(* Logix 5000 project; controller APM_Sopladora Emulate 5570 rev 32.11; software revision 32.00 *)

TASK MainTask (continuous, watchdog 500 ms) : MainProgram

MODULES
   Local : Emulate 5570 (ICP 2, rev 32.11)
END_MODULES

VAR_GLOBAL   (* controller tags *)
   A_AbrirMoldes : BOOL;
   A_BandaSopladora : BOOL;
   A_Bandeja : BOOL;
   A_BrazoEx : BOOL;
   A_Grib : BOOL;
   A_Piston : BOOL;
   Aux_Grib : BOOL;
   Aux_Puerta : BOOL;
   BaGF : BOOL;
   BaGF_Ok : BOOL;
   BaGR : BOOL;
   BaGR_Ok : BOOL;
   BaMF : BOOL;
   BaMF_Ok : BOOL;
   BaMR : BOOL;
   BaMR_Ok : BOOL;
   CA_BorrarBotPre : BOOL;
   CA_BotFin : BOOL;
   CA_BotPre : BOOL;
   Count : COUNTER := (PRE := 5);
   Etapa1 : BOOL;
   Etapa10 : BOOL;
   Etapa11 : BOOL;
   Etapa12 : BOOL;
   Etapa13 : BOOL;
   Etapa1A : BOOL;
   Etapa2 : BOOL;
   Etapa2A : BOOL;
   Etapa3 : BOOL;
   Etapa4 : BOOL;
   Etapa5 : BOOL;
   Etapa6 : BOOL;
   Etapa7 : BOOL;
   Etapa8 : BOOL;
   Etapa9 : BOOL;
   Etapa9A : BOOL;
   ND_Start : BOOL;
   ND_Stop : BOOL;
   S_BandejaAtras : BOOL;
   S_BandejaFrente : BOOL;
   S_BotAtGrip : BOOL;
   S_BotAtMolde : BOOL;
   S_BrazoExtendido : BOOL;
   S_BrazoRecogido : BOOL;
   S_PistonAbajo : BOOL;
   S_PistonArriba : BOOL;
   S_PuertaAbierta : BOOL;
   S_PuertaCerrada : BOOL;
   S_Salida : BOOL;
   Sal : BOOL;
   Sal_Ok : BOOL;
   Sec : BOOL;
   Timer1 : TIMER := (PRE := 5000);
   Timer2 : TIMER := (PRE := 3000);
   Timer3 : TIMER := (PRE := 4000);
END_VAR

PROGRAM MainProgram   (* main routine MainRoutine *)

ROUTINE MainRoutine   (* ladder *)
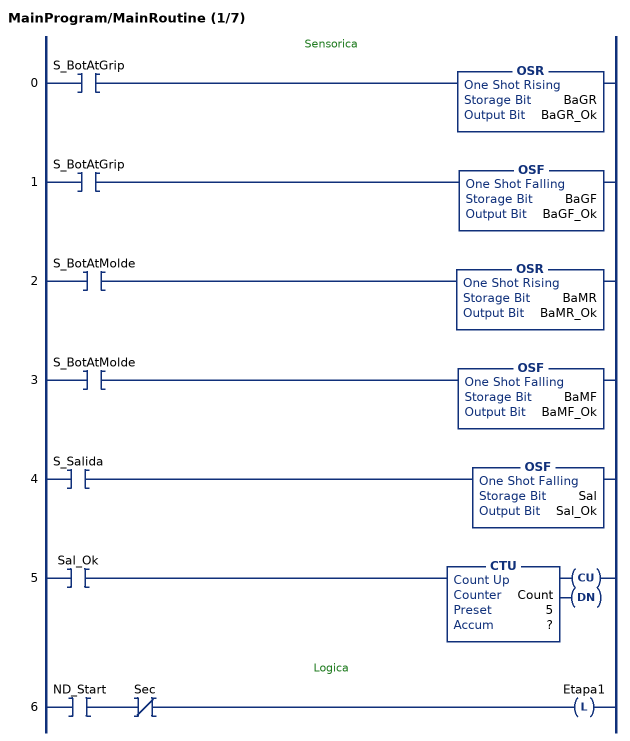
   // Sensorica
   0: XIC(S_BotAtGrip)OSR(BaGR,BaGR_Ok);
   1: XIC(S_BotAtGrip)OSF(BaGF,BaGF_Ok);
   2: XIC(S_BotAtMolde)OSR(BaMR,BaMR_Ok);
   3: XIC(S_BotAtMolde)OSF(BaMF,BaMF_Ok);
   4: XIC(S_Salida)OSF(Sal,Sal_Ok);
   5: XIC(Sal_Ok)CTU(Count,?,?);
   // Logica
   6: XIC(ND_Start)XIO(Sec)OTL(Etapa1);
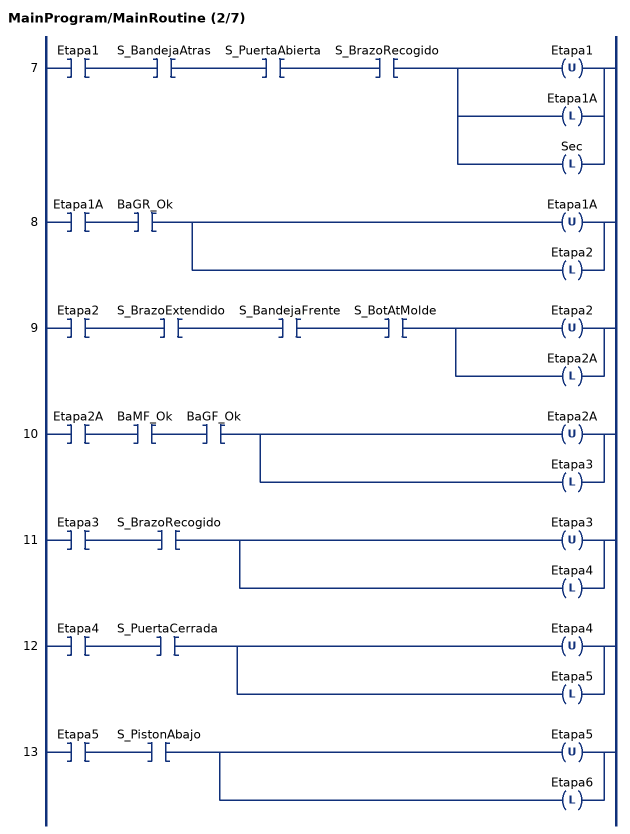
   7: XIC(Etapa1)XIC(S_BandejaAtras)XIC(S_PuertaAbierta)XIC(S_BrazoRecogido)[OTU(Etapa1) ,[OTL(Etapa1A) ,OTL(Sec) ] ];
   8: XIC(Etapa1A)XIC(BaGR_Ok)[OTU(Etapa1A) ,OTL(Etapa2) ];
   9: XIC(Etapa2)XIC(S_BrazoExtendido)XIC(S_BandejaFrente)XIC(S_BotAtMolde)[OTU(Etapa2) ,OTL(Etapa2A) ];
   10: XIC(Etapa2A)XIC(BaMF_Ok)XIC(BaGF_Ok)[OTU(Etapa2A) ,OTL(Etapa3) ];
   11: XIC(Etapa3)XIC(S_BrazoRecogido)[OTU(Etapa3) ,OTL(Etapa4) ];
   12: XIC(Etapa4)XIC(S_PuertaCerrada)[OTU(Etapa4) ,OTL(Etapa5) ];
   13: XIC(Etapa5)XIC(S_PistonAbajo)[OTU(Etapa5) ,OTL(Etapa6) ];
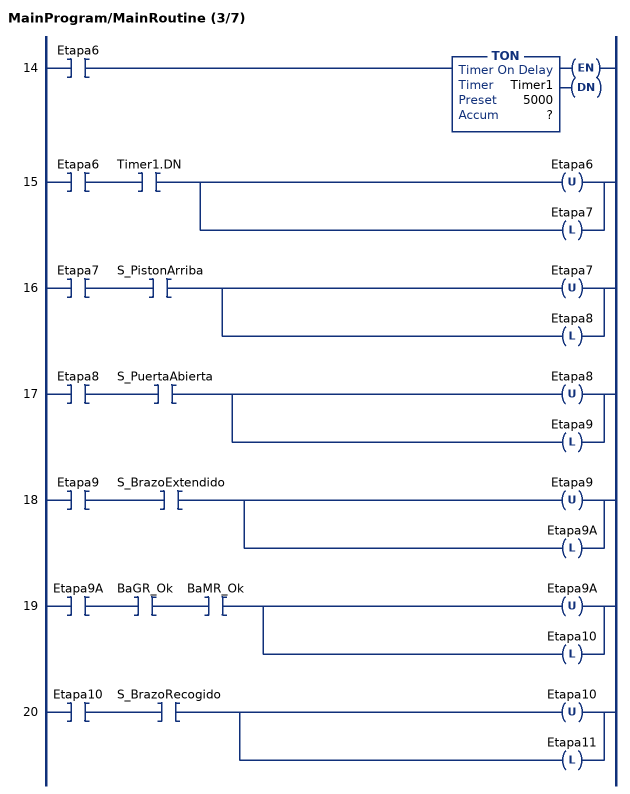
   14: XIC(Etapa6)TON(Timer1,?,?);
   15: XIC(Etapa6)XIC(Timer1.DN)[OTU(Etapa6) ,OTL(Etapa7) ];
   16: XIC(Etapa7)XIC(S_PistonArriba)[OTU(Etapa7) ,OTL(Etapa8) ];
   17: XIC(Etapa8)XIC(S_PuertaAbierta)[OTU(Etapa8) ,OTL(Etapa9) ];
   18: XIC(Etapa9)XIC(S_BrazoExtendido)[OTU(Etapa9) ,OTL(Etapa9A) ];
   19: XIC(Etapa9A)XIC(BaGR_Ok)XIC(BaMR_Ok)[OTU(Etapa9A) ,OTL(Etapa10) ];
   20: XIC(Etapa10)XIC(S_BrazoRecogido)[OTU(Etapa10) ,OTL(Etapa11) ];
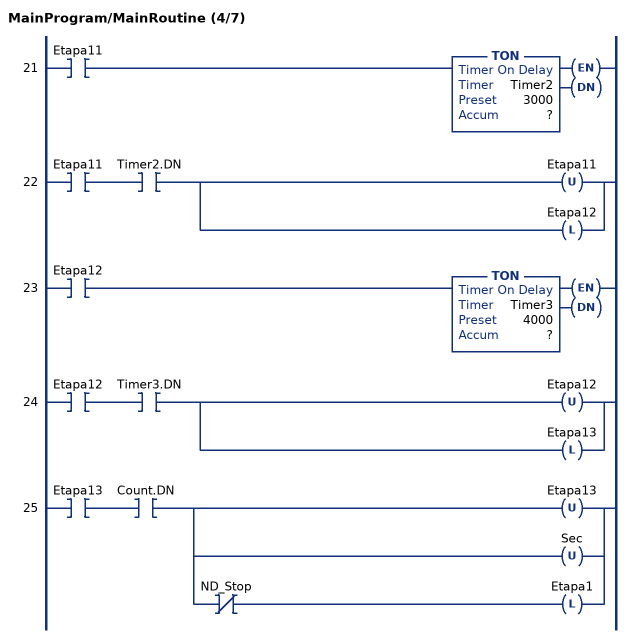
   21: XIC(Etapa11)TON(Timer2,?,?);
   22: XIC(Etapa11)XIC(Timer2.DN)[OTU(Etapa11) ,OTL(Etapa12) ];
   23: XIC(Etapa12)TON(Timer3,?,?);
   24: XIC(Etapa12)XIC(Timer3.DN)[OTU(Etapa12) ,OTL(Etapa13) ];
   25: XIC(Etapa13)XIC(Count.DN)[OTU(Etapa13) ,[OTU(Sec) ,XIO(ND_Stop) OTL(Etapa1) ] ];
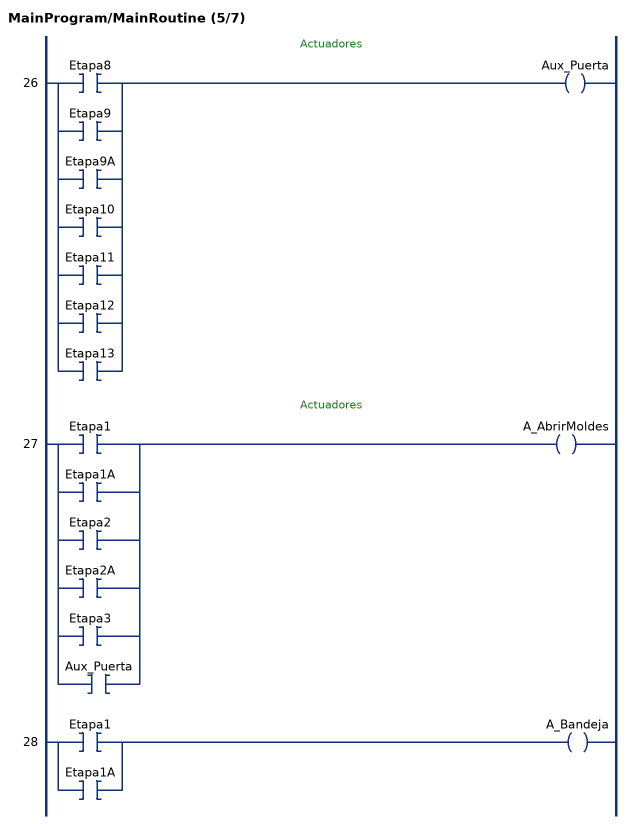
   // Actuadores
   26: [XIC(Etapa8) ,[XIC(Etapa9) ,[XIC(Etapa9A) ,[XIC(Etapa10) ,[XIC(Etapa11) ,[XIC(Etapa12) ,XIC(Etapa13) ] ] ] ] ] ]OTE(Aux_Puerta);
   // Actuadores
   27: [XIC(Etapa1) ,[XIC(Etapa1A) ,[XIC(Etapa2) ,[XIC(Etapa2A) ,[XIC(Etapa3) ,XIC(Aux_Puerta) ] ] ] ] ]OTE(A_AbrirMoldes);
   28: [XIC(Etapa1) ,XIC(Etapa1A) ]OTE(A_Bandeja);
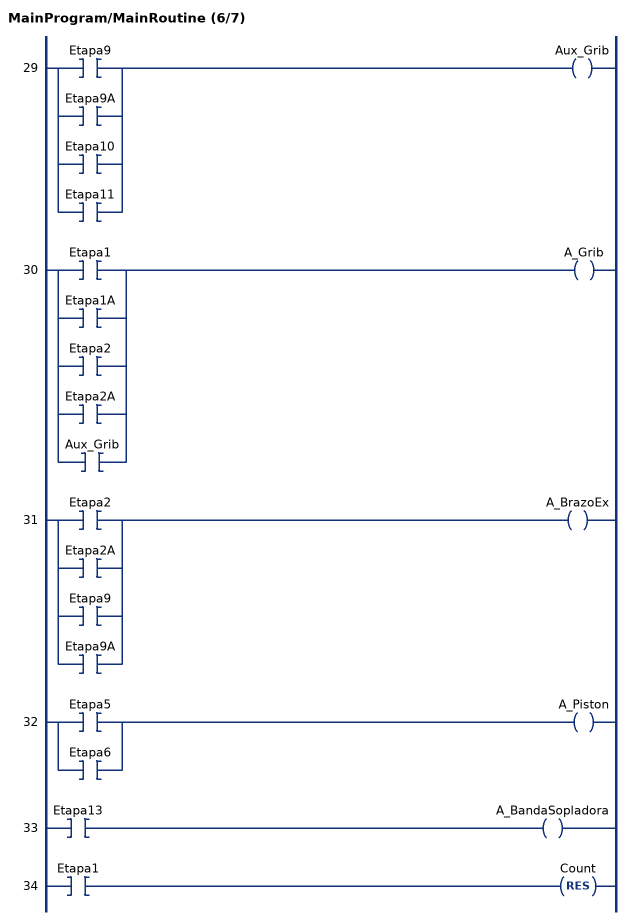
   29: [XIC(Etapa9) ,[XIC(Etapa9A) ,[XIC(Etapa10) ,XIC(Etapa11) ] ] ]OTE(Aux_Grib);
   30: [XIC(Etapa1) ,[XIC(Etapa1A) ,[XIC(Etapa2) ,[XIC(Etapa2A) ,XIC(Aux_Grib) ] ] ] ]OTE(A_Grib);
   31: [XIC(Etapa2) ,[XIC(Etapa2A) ,[XIC(Etapa9) ,XIC(Etapa9A) ] ] ]OTE(A_BrazoEx);
   32: [XIC(Etapa5) ,XIC(Etapa6) ]OTE(A_Piston);
   33: XIC(Etapa13)OTE(A_BandaSopladora);
   34: XIC(Etapa1)RES(Count);
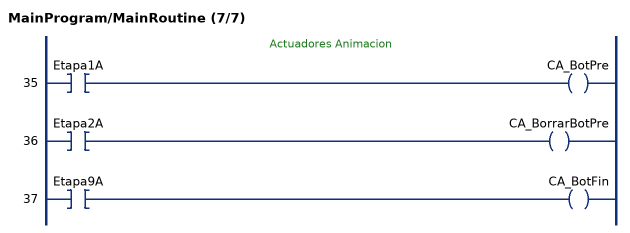
   // Actuadores Animacion
   35: XIC(Etapa1A)OTE(CA_BotPre);
   36: XIC(Etapa2A)OTE(CA_BorrarBotPre);
   37: XIC(Etapa9A)OTE(CA_BotFin);
END_ROUTINE
END_PROGRAM
